// TIA Portal V19 export
VAR_GLOBAL   // PLC tag table "U2Em0"
END_VAR
